PROGRAM MAIN
VAR
END_VAR

fbStation();

GVL.stParam.stStatus.lrPositionMoteur:=GVL.axeX.NcToPlc.ActPos;

GVL.stIO.stOut.xMotPosBasse:=GVL.axeX.NcToPlc.ActPos<=GVL.stParam.stRecipe.lrPositionBasse+0.01;

GVL.stIO.stOut.xMotPosHaute:=GVL.axeX.NcToPlc.ActPos>=-0.01;

END_PROGRAM

(* stored: Version 1.1.0.1, ProductVersion 3.1.4020.12
   POU MAIN: Id {8bc51daa-5a89-48e9-a5c4-d77fc3d52b56}, SpecialFunc None *)
